Fanuc KAREL source: kd00021.KL

-- PROVISIONAL review KL for V940-1; original PC SHA256 12e6633c65e21099d36afeecfedcedf058add22906cecd9a245c5e6b61482dc5
-- Incomplete behavior may be omitted. Consult companion uncertainty JSON. Do not deploy.
PROGRAM KD00021
%NOLOCKGROUP
BEGIN
  -- V9_ZERO_TABLE_METADATA_HINT layout=0002_ascii; no indexed target words; source/name/runtime held
  -- UNRESOLVED_PC offsets 5-17; opcodes 21,23
  -- UNRESOLVED_PC offsets 22-26; opcodes 7F
END KD00021
